FUNCTION_BLOCK FalseBoolValue IMPLEMENTS BoolValue
VAR
END_VAR

{attribute 'monitoring' := 'call'}
PROPERTY Value : BOOL
GET
Value := FALSE;
END_GET
END_PROPERTY

END_FUNCTION_BLOCK

(* stored: Version 1.1.0.1
   POU FalseBoolValue: Id {4cc27881-c1fe-4640-b030-93443251dfce}, SpecialFunc None
   Property Value: Id {4a467719-df03-4b51-a941-213ea6ab9e51}
   Get Get: Id {a056c52a-b0cb-43c6-9486-ed882b0d9ac2} *)
